GLOBALCONSTANTS DataPanel_MI_AQ (* DataPanel Modules with medium IO density AQ constants *)
  (* Standard: 61499-1; Description: Copyright (c) 2026 HR Agrartechnik GmbH *)
  (* Version 1.0, 2026-01-16, generated, HR Agrartechnik GmbH *)
  PACKAGE DataPanel::io::MI::AQ;
  VAR_GLOBAL CONSTANT
    AnalogOutput_1A : DataPanel::io::MI::AQ::DataPanel_MI_AQ_S := (Pin := 1);
    AnalogOutput_1B : DataPanel::io::MI::AQ::DataPanel_MI_AQ_S := (Pin := 2);
    AnalogOutput_2A : DataPanel::io::MI::AQ::DataPanel_MI_AQ_S := (Pin := 3);
    AnalogOutput_2B : DataPanel::io::MI::AQ::DataPanel_MI_AQ_S := (Pin := 4);
    AnalogOutput_3A : DataPanel::io::MI::AQ::DataPanel_MI_AQ_S := (Pin := 5);
    AnalogOutput_3B : DataPanel::io::MI::AQ::DataPanel_MI_AQ_S := (Pin := 6);
    AnalogOutput_4A : DataPanel::io::MI::AQ::DataPanel_MI_AQ_S := (Pin := 7);
    AnalogOutput_4B : DataPanel::io::MI::AQ::DataPanel_MI_AQ_S := (Pin := 8);
    AnalogOutput_5A : DataPanel::io::MI::AQ::DataPanel_MI_AQ_S := (Pin := 9);
    AnalogOutput_5B : DataPanel::io::MI::AQ::DataPanel_MI_AQ_S := (Pin := 10);
    AnalogOutput_6A : DataPanel::io::MI::AQ::DataPanel_MI_AQ_S := (Pin := 11);
    AnalogOutput_6B : DataPanel::io::MI::AQ::DataPanel_MI_AQ_S := (Pin := 12);
    AnalogOutput_7A : DataPanel::io::MI::AQ::DataPanel_MI_AQ_S := (Pin := 13);
    AnalogOutput_7B : DataPanel::io::MI::AQ::DataPanel_MI_AQ_S := (Pin := 14);
    AnalogOutput_8A : DataPanel::io::MI::AQ::DataPanel_MI_AQ_S := (Pin := 15);
    AnalogOutput_8B : DataPanel::io::MI::AQ::DataPanel_MI_AQ_S := (Pin := 16);
    Invalid : DataPanel::io::MI::AQ::DataPanel_MI_AQ_S := (Pin := 255);
  END_VAR
END_GLOBALCONSTANTS
